{attribute 'qualified_only'}
VAR_GLOBAL
	// ATM: 2 Axes
    {attribute 'pytmc' := 'pv: MFX:ATM:MMS:Y'}
    //{attribute 'TcLinkTo' := '.bLimitForwardEnable  := TIIB[MFX-ATM-EL7041-E1]^STM Status^Status^Digital input 1;
    //                          .bLimitBackwardEnable := TIIB[MFX-ATM-EL7041-E1]^STM Status^Status^Digital input 2;
    //                          .bBrakeRelease        := TIIB[MFX-ATM-EL2004-E4]^Channel 1^Output;
    //                          .nRawEncoderULINT     := TIIB[MFX-ATM-EL5042-E3]^FB Inputs Channel 1^Position'}
	{attribute 'TcLinkTo' := '.bLimitForwardEnable  := TIIB[MFX-ATM-EL7041-E1]^STM Status^Status^Digital input 1;
                              .bLimitBackwardEnable := TIIB[MFX-ATM-EL7041-E1]^STM Status^Status^Digital input 2;
                              .nRawEncoderULINT     := TIIB[MFX-ATM-EL5042-E3]^FB Inputs Channel 1^Position'}
    M1: DUT_MotionStage := (sName := 'MFX:ATM:MMS:Y');
    {attribute 'pytmc' := 'pv: MFX:ATM:MMS:X'}
    {attribute 'TcLinkTo' := '.nRawEncoderULINT     := TIIB[MFX-ATM-EL5042-E3]^FB Inputs Channel 2^Position'}
    M2: DUT_MotionStage := (sName := 'MFX:ATM:MMS:X');
	
	
    // LIB-: 4 Axes
    {attribute 'pytmc' := 'pv: MFX:LIB:MMS:01'}
	{attribute 'TcLinkTo' := '.bLimitForwardEnable  := TIIB[MFX-LIB-EL1088-E5]^Channel 1^Input;
                              .bLimitBackwardEnable := TIIB[MFX-LIB-EL1088-E5]^Channel 2^Input'}
    M3: DUT_MotionStage := (sName := 'MFX:LIB:MMS:01');
	{attribute 'pytmc' := 'pv: MFX:LIB:MMS:02'}
	{attribute 'TcLinkTo' := '.bLimitForwardEnable  := TIIB[MFX-LIB-EL1088-E5]^Channel 3^Input;
                              .bLimitBackwardEnable := TIIB[MFX-LIB-EL1088-E5]^Channel 4^Input'}
	M4: DUT_MotionStage := (sName := 'MFX:LIB:MMS:02');
	{attribute 'pytmc' := 'pv: MFX:LIB:MMS:03'}
	{attribute 'TcLinkTo' := '.bLimitForwardEnable  := TIIB[MFX-LIB-EL1088-E5]^Channel 5^Input;
                              .bLimitBackwardEnable := TIIB[MFX-LIB-EL1088-E5]^Channel 6^Input'}
	M5: DUT_MotionStage := (sName := 'MFX:LIB:MMS:03');
	{attribute 'pytmc' := 'pv: MFX:LIB:MMS:04'}
	{attribute 'TcLinkTo' := '.bLimitForwardEnable  := TIIB[MFX-LIB-EL1088-E5]^Channel 7^Input;
                              .bLimitBackwardEnable := TIIB[MFX-LIB-EL1088-E5]^Channel 8^Input'}
	M6: DUT_MotionStage := (sName := 'MFX:LIB:MMS:04');
    
    // LJ-: 8 Axes

	{attribute 'pytmc' := 'pv: MFX:LJH:JET:X'}
	{attribute 'TcLinkTo' := '.bLimitForwardEnable  := TIIB[MFX-LJ-EL1088-E3]^Channel 1^Input;
                              .bLimitBackwardEnable := TIIB[MFX-LJ-EL1088-E3]^Channel 2^Input'}
    M7: DUT_MotionStage := (sName := 'MFX:LJH:JET:X');

	{attribute 'pytmc' := 'pv: MFX:LJH:JET:Y'}
	{attribute 'TcLinkTo' := '.bLimitForwardEnable  := TIIB[MFX-LJ-EL1088-E3]^Channel 4^Input;
                              .bLimitBackwardEnable := TIIB[MFX-LJ-EL1088-E3]^Channel 3^Input'}
    M8: DUT_MotionStage := (sName := 'MFX:LJH:JET:Y');

	{attribute 'pytmc' := 'pv: MFX:LJH:JET:Z'}
	{attribute 'TcLinkTo' := '.bLimitForwardEnable  := TIIB[MFX-LJ-EL1088-E8]^Channel 1^Input;
                              .bLimitBackwardEnable := TIIB[MFX-LJ-EL1088-E8]^Channel 2^Input'}
    M9: DUT_MotionStage := (sName := 'MFX:LJH:JET:Z');
    
	{attribute 'pytmc' := 'pv: MFX:LJH:DET:X'}
	{attribute 'TcLinkTo' := '.bLimitForwardEnable  := TIIB[MFX-LJ-EL1088-E8]^Channel 3^Input;
                              .bLimitBackwardEnable := TIIB[MFX-LJ-EL1088-E8]^Channel 4^Input'}
    M10: DUT_MotionStage := (sName := 'MFX:LJH:DET:X');

	{attribute 'pytmc' := 'pv: MFX:LJH:SS:TOP_X'}
	{attribute 'TcLinkTo' := '.bLimitForwardEnable  := TIIB[MFX-LJ-EL1088-E12]^Channel 1^Input;
                              .bLimitBackwardEnable := TIIB[MFX-LJ-EL1088-E12]^Channel 2^Input'}
    M11: DUT_MotionStage := (sName := 'MFX:LJH:SS:TOP_X');

	{attribute 'pytmc' := 'pv: MFX:LJH:SS:TOP_Y'}
	{attribute 'TcLinkTo' := '.bLimitForwardEnable  := TIIB[MFX-LJ-EL1088-E12]^Channel 3^Input;
                              .bLimitBackwardEnable := TIIB[MFX-LJ-EL1088-E12]^Channel 4^Input'}
    M12: DUT_MotionStage := (sName := 'MFX:LJH:SS:TOP_Y');

	{attribute 'pytmc' := 'pv: MFX:LJH:SS:BOT_X'}
	{attribute 'TcLinkTo' := '.bLimitForwardEnable  := TIIB[MFX-LJ-EL1088-E12]^Channel 5^Input;
                              .bLimitBackwardEnable := TIIB[MFX-LJ-EL1088-E12]^Channel 6^Input'}
    M13: DUT_MotionStage := (sName := 'MFX:LJH:SS:BOT_X');

	{attribute 'pytmc' := 'pv: MFX:LJH:SS:BOT_Y'}
	{attribute 'TcLinkTo' := '.bLimitForwardEnable  := TIIB[MFX-LJ-EL1088-E12]^Channel 7^Input;
                              .bLimitBackwardEnable := TIIB[MFX-LJ-EL1088-E12]^Channel 8^Input'}
    M14: DUT_MotionStage := (sName := 'MFX:LJH:SS:BOT_Y');
END_VAR

(* stored: Version 1.1.0.1, ProductVersion 3.1.4022.18
   GVL Main: Id {1691e643-5c47-48e9-bb1a-9f3fc0d078a1} *)
